FUNCTION_BLOCK EL2024
VAR
	{attribute addProperty Name "WcState"}
	_wcState : WcStateBase;
	{attribute addProperty Name "Info data"}
	_infoData : InfoDataBase;
	_io : EL2xx4_Data;
END_VAR

PROPERTY IO : REFERENCE TO EL2xx4_Data
GET
IO REF= _io;
END_GET
END_PROPERTY

PROPERTY WcState : REFERENCE TO WcStateBase
GET
WcState REF= _wcState;
END_GET
END_PROPERTY

END_FUNCTION_BLOCK

(* stored: Version 1.1.0.1, ProductVersion 3.1.4024.9
   POU EL2024: Id {e608f0f1-b53b-0701-2b2d-0d5bd2452e45}, SpecialFunc None
   Property IO: Id {109fc22b-3fe4-0771-120e-44dd8c8ead94}
   Get Get: Id {07570e0d-a92f-02af-1fa7-1ab295464f24}
   Property WcState: Id {3fe43c3f-7120-0d11-20d1-3f6dd876ca06}
   Get Get: Id {da747640-b2e1-0841-2171-8595d547f4fc} *)
